TYPE U_FilterThickness :
UNION
    fThickness : LREAL; // [mm]
    stWedge : ST_Wedge;
END_UNION
END_TYPE

(* stored: Version 1.1.0.1
   DUT U_FilterThickness: Id {15675aa2-30d7-46ca-8829-d58b11d473fd} *)
